# EPICS autosave request: testApp/Db/TISCamMenu.req
file "configMenu.req", P=$(P), CONFIG=$(CONFIG)
file "configMenu_settings.req", P=$(P), CONFIG=$(CONFIG)
file "aravisCamera_settings.req", P=$(P), R=cam1:
